// TIA Portal V19 export
FUNCTION "BIT_COUNT" : Int   // FC6, LAD
TITLE = BIT COUNT
// stored: SetENOAutomatically false
   VAR_INPUT
      Data : Variant;
   END_VAR
   VAR_TEMP
      i : ULInt;
      BitNumber : ULInt;
      LocalByte : Byte;
      LocalWord : Word;
      LocalInt : Int;
      LocalDWord : DWord;
      LocalDint : DInt;
      DataToCheck : DWord;
      Result : DWord;
      retVal : Int;
   END_VAR
BEGIN

REGION Network 1 (SCL): Detect
   IF  TypeOf(#Data) = Byte THEN
       #BitNumber := 8;
       #retVal := MOVE_BLK_VARIANT(SRC:=#Data, COUNT:=1, SRC_INDEX:=0, DEST_INDEX:=0, DEST=>#LocalByte);
       #DataToCheck := #LocalByte;
   ELSIF TypeOf(#Data) = Word THEN
       #BitNumber := 16;
       #retVal := MOVE_BLK_VARIANT(SRC:=#Data, COUNT:=1, SRC_INDEX:=0, DEST_INDEX:=0, DEST=>#LocalWord);
       #DataToCheck := #LocalWord;
   ELSIF TypeOf(#Data) = Int THEN
       #BitNumber := 16;
       #retVal := MOVE_BLK_VARIANT(SRC:=#Data, COUNT:=1, SRC_INDEX:=0, DEST_INDEX:=0, DEST=>#LocalInt);
       #DataToCheck := INT_TO_DWORD(#LocalInt);
   ELSIF TypeOf(#Data) = DWord THEN
       #BitNumber := 32;
       #retVal := MOVE_BLK_VARIANT(SRC:=#Data, COUNT:=1, SRC_INDEX:=0, DEST_INDEX:=0, DEST=>#LocalDWord);
       #DataToCheck := #LocalDWord;
   ELSIF TypeOf(#Data) = DInt THEN
       #BitNumber := 32;
       #retVal := MOVE_BLK_VARIANT(SRC:=#Data, COUNT:=1, SRC_INDEX:=0, DEST_INDEX:=0, DEST=>#LocalDint);
       #DataToCheck := DINT_TO_DWORD(#LocalDint);
   ELSE
       #BitNumber := 0;
   END_IF;

   #BIT_COUNT := 0;

   IF #BitNumber > 0 THEN
       //Count data
       FOR #i := 0 TO #BitNumber -1 DO
           #Result := SHR(IN:=#DataToCheck, N:=#i);
           IF #Result.%X0 THEN
               #BIT_COUNT +=1;
           END_IF;
       END_FOR;
   END_IF;
END_REGION
END_FUNCTION
